(* PLC project Tc2_Utilities.F_GetDOYOfYearMonthDay Demo, tc3-libraries-kb TwinCAT 3.1 *)
(* stored: creationDateTime 2026-05-11T12:00:00, modificationDateTime 2026-05-11T12:00:00 *)

PROGRAM P_Demo_F_GetDOYOfYearMonthDay
  VAR
    wYear : WORD := 2026;  (* 年份 *)
    wMonth : WORD := 5;  (* 月 *)
    wDay : WORD := 11;  (* 日 *)
    wDOY : WORD;  (* 年内第几天（1~366） *)
    bRunOnce : BOOL;  (* 脉冲触发 *)
  END_VAR

// =============================================================================
// 场景：太阳能 / 气象模型按「年内第几天」(DOY) 做日辐射强度查表
//
// 价值：1 行调用避免手写「累加各月天数 + 闰年判定」，特别是 2 月闰年规则
//
// 验证步骤：
//   1. 引用 Tc2_Utilities
//   2. 编译 + 登录 + 运行
//   3. 强制 bRunOnce := TRUE
//   4. 在线观察 wDOY 应为 131（2026 年 5 月 11 日是第 131 天）
//   5. wMonth:=2, wDay:=29; wYear:=2024 → wDOY = 60（闰年 2 月 29 是第 60 天）
//   6. wYear:=2023 同条件 → wDOY = 0（平年没有 2 月 29 日）
// =============================================================================
wDOY := F_GetDOYOfYearMonthDay(wYear, wMonth, wDay);
END_PROGRAM
